(* CoDeSys 2.3.9.41 project: lek_temp80_1.pro *)
(* Libraries: Standard.lib 4.10.05 11:14:46, IecSfc.lib 13.4.06 15:51:28, SYSLIBCALLBACK.LIB 26.9.08 16:43:52 *)

(* POU PLC_PRG, ST *)
PROGRAM PLC_PRG
VAR
	Tempmin:REAL:=0;
	Tempmax:REAL:=0;
	Tokmin:REAL:=0;
	Tokmax:REAL:=0;
	Temp : REAL; (*температура*)
	Tok : REAL; (*ток 4-20 мА*)
	lamp1: BOOL; (*лампа, выход за диапазон 0-80 градусов*)
END_VAR
IF (Tempmin <> Tempmax) THEN

Tok:=(Tokmax-Tokmin)*((Temp-Tempmin)/(Tempmax-Tempmin))+Tokmin;
ELSE
Tok:=0;
END_IF



(* lamp1 := (Temp1 > 80.0)  OR (Temp1 < 0) ;
Prom := LIMIT (0 , Temp1 , 80);
Tok := (( 16.0 / 80 ) * Prom ) + 4.0 ; *)
END_PROGRAM
